# B&R Automation Studio project AnsteuerungSchrittmotor
Automation Studio 4.3.7.46 SP; technology packages: Acp10Arnc0 3.18.2

## Configuration Config1

CPU 4PP065.0571-P74, AutomationRuntime G4.34, Build 4.1.2, Vc V4.34.3

### Hardware
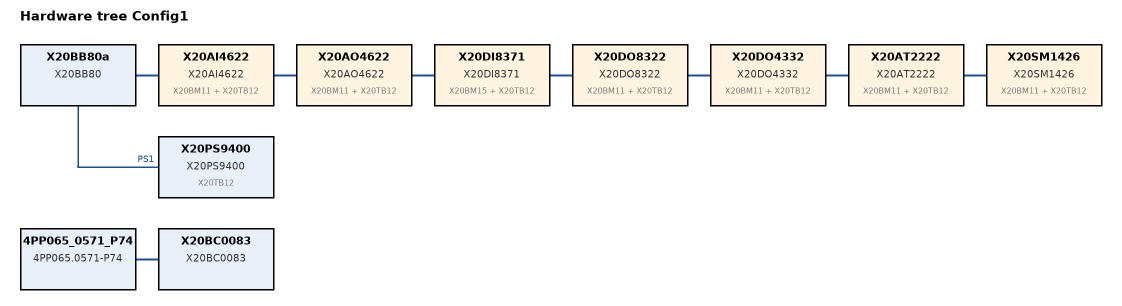
```
4PP065_0571_P74 : 4PP065.0571-P74 v1.1.2.0
  Connector IF5:
    ActivateDevice = 1
    Mode = Manual
    InternetAddress = 10.100.85.8
    SubnetMask = 255.255.255.0
  ConfigurationID = KainerKerschbaumer_Config1
  TimerDeviceType = EPLX2X
  TimerDevice = 4PP065_0571_P74.IF4
  TaskClassIdleTime = 2000
  Cyclic1Duration = 2000
  Cyclic1Tolerance = 0
  Cyclic1Output = 1
  VcObjectName = Visu
X20AI4622 : X20AI4622 v1.0.4.0  [SS1 -> X20TB12.SS; SL -> X20BM11.SL1]
X20AO4622 : X20AO4622 v1.1.0.0  [SS1 -> X20TB12e.SS; SL -> X20BM11c.SL1]
X20AT2222 : X20AT2222 v1.2.1.0  [SS1 -> X20TB12f.SS; SL -> X20BM11d.SL1]
X20BB80a : X20BB80 v1.0.1.0
X20BC0083 : X20BC0083 v2.5.3.0  [PLK1 -> 4PP065_0571_P74.IF4 (NodeNumber=1) [Cable Type=PowerlinkCable, Length=10, Version=1.0.0.1]; SL -> X20BB80a.SL1]
X20BM11 : X20BM11 v1.0.0.1  [X2X1 -> X20BB80a.IF1]
X20BM11a : X20BM11 v1.0.0.1  [X2X1 -> X20BM15.X2X2]
X20BM11b : X20BM11 v1.0.0.1  [X2X1 -> X20BM11a.X2X2]
X20BM11c : X20BM11 v1.0.0.1  [X2X1 -> X20BM11.X2X2]
X20BM11d : X20BM11 v1.0.0.1  [X2X1 -> X20BM11b.X2X2]
X20BM11e : X20BM11 v1.0.0.1  [X2X1 -> X20BM11d.X2X2]
X20BM15 : X20BM15 v1.0.1.0  [X2X1 -> X20BM11c.X2X2 (NodeNumber=4)]
X20DI8371 : X20DI8371 v1.0.2.0  [SS1 -> X20TB12a.SS; SL -> X20BM15.SL1]
X20DO4332 : X20DO4332 v1.0.3.0  [SS1 -> X20TB12d.SS; SL -> X20BM11b.SL1]
X20DO8322 : X20DO8322 v1.0.2.0  [SS1 -> X20TB12c.SS; SL -> X20BM11a.SL1]
X20PS9400 : X20PS9400 v1.0.2.4  [SS1 -> X20TB12b.SS; PS -> X20BB80a.PS1]
X20SM1426 : X20SM1426 v1.5.1.1  [SS1 -> X20TB12g.SS; SL -> X20BM11e.SL1]
  HoldingCurrent = 60
  RatedCurrent = 80
  MaximumCurrent = 100
  LatchSync = Stepper latch value synchron (AB/R latch value asynchron)
  SCALE_ENCOD_INCR_r1 = 51200
  BothEndSwitchesAreNormallyOpen_r1 = on
  QuickStopIsNormallyOpen_r1 = on
X20TB12 : X20TB12 v1.0.0.0
X20TB12a : X20TB12 v1.0.0.0
X20TB12b : X20TB12 v1.0.0.0
X20TB12c : X20TB12 v1.0.0.0
X20TB12d : X20TB12 v1.0.0.0
X20TB12e : X20TB12 v1.0.0.0
X20TB12f : X20TB12 v1.0.0.0
X20TB12g : X20TB12 v1.0.0.0
```

### IoMap.iom - 4PP065_0571_P74/IoMap.iom
```iecst
VAR_CONFIG
	       Cyclic#1.gAxis01_DrvIf.iLifeCnt AT %IB."X20SM1426".LifeCnt;
	       Cyclic#1.gAxis01_DrvIf.iDrvOK AT %IX."X20SM1426".DrvOk01;
	       Cyclic#1.gAxis01_DrvIf.oBoostCurrent AT %QX."X20SM1426".BoostCurrent01;
	       Cyclic#1.gAxis01_DrvIf.oStandStillCurrent AT %QX."X20SM1426".StandstillCurrent01;
	       Cyclic#1.gAxis01_DrvIf.oSetTime AT %QW."X20SM1426".SetTime01;
	       Cyclic#1.gAxis01_MotorStep0 AT %QW."X20SM1426".Motor1Step0;
	       Cyclic#1.gAxis01_DiDoIf.iLifeCntDriveEnable AT %IB."X20SM1426".LifeCnt;
	       Cyclic#1.gAxis01_DiDoIf.iLifeCntDriveReady AT %IB."X20SM1426".LifeCnt;
	       Cyclic#1.gAxis01_DiDoIf.iDriveReady AT %IX."X20SM1426".DrvOk01;
	       Cyclic#1.gAxis01_DiDoIf.oDriveEnable AT %QX."X20SM1426".DriveEnable01;
	       Cyclic#1.gAxis01_EncIf1.iLifeCnt AT %IB."X20SM1426".LifeCnt;
	       Cyclic#1.gAxis01_EncIf1.iEncOK AT %IX."X20SM1426".EncOk01;
	       Cyclic#1.gAxis01_EncIf1.iActPos AT %IW."X20SM1426".ActPos01;
	       Cyclic#1.gAxis01_EncIf1.iRefPulsePos AT %IW."X20SM1426".RefPulsePos01;
	       Cyclic#1.gAxis01_EncIf1.iRefPulseCnt AT %IB."X20SM1426".RefPulseCnt01;
	       Cyclic#1.gAxis01_EncIf1.iActTime AT %IW."X20SM1426".ActTime01;
END_VAR
```

### Acp10cfg.ncc - 4PP065_0571_P74/Motion/Acp10cfg.ncc
```
NcConfiguration (Version=3.18.2, NcSwId=Acp10)
  ACP10CF1_typ:
    cnt_nettrc_rec_drive = 1500
    bufsize_trace_upload = 1200
    tc_nc_man_task = Cyclic #1
    glob_pv_as_ncobject = Yes
    ncsys_dl_broadcast = Yes
    ncsys_dl_acp_reset = Yes
    safemc_log_err_to_ax = Yes
    network_init:
      ncsw_init_execute = Yes
      automatic_execute = No
      node_nr_warning = Yes
      net_err_before_ncact = Yes
    nettrc:
      enter_parsecrec = Yes
      enter_ncaction = Yes
      save_ring_startidx = Yes
    cam_prof_download:
      cam_dat_dl_parallel = No
      tc_cam_dl_parallel = Task class for NC Manager task
    sdc_if[0]:
      if_name = SDC_IF1
      mc_broadcast_size = 800
      mc_broadcast_extdat = No
```

### Acp10map.ncm - 4PP065_0571_P74/Motion/Acp10map.ncm
```
NcMapping (NcSwId=Acp10)
  NcObject gAxis01 (ModuleId=X20SM1426, ModuleAddress=SDC_IF1.ST1, Type=ncAXIS, Channel=1, AcoposSimulation=Off, InitParameter=gAxis01i, AcoposParameter=gAxis01a, Disabled=FALSE, ModuleDisabled=FALSE)
```

## Logical view

Binary libraries used (declarations not repeated): operator, runtime, astime, AsIecCon, Acp10man 3.18.2, Acp10par 3.18.2, NcGlobal 3.18.2, Acp10sdc 3.18.2, Acp10_MC 3.18.2, brsystem, sys_lib, AsBrStr

### Global.var - Global variables
```iecst
VAR
	gAxis01 : ACP10AXIS_typ;
	gAxis01_HW : SdcHwCfg_typ := (0);
	gAxis01_DrvIf : SdcDrvIf16_typ := (0);
	gAxis01_EncIf1 : SdcEncIf16_typ := (0);
	gAxis01_DiDoIf : SdcDiDoIf_typ := (0);
	gAxis01_MotorStep0 : INT := (0);
END_VAR
```


### Program Logical/ncsdcctrl (IEC)

#### ncsdcctrlCyclic.st
```iecst
PROGRAM _CYCLIC

(* ### BEGIN gAxis01 ### *)

(* life counter emulation of digital inputs *)
       gAxis01_DiDoIf.iLifeCntReference := gAxis01_DiDoIf.iLifeCntReference + 1;
       gAxis01_DiDoIf.iLifeCntNegHwEnd  := gAxis01_DiDoIf.iLifeCntNegHwEnd  + 1;
       gAxis01_DiDoIf.iLifeCntPosHwEnd  := gAxis01_DiDoIf.iLifeCntPosHwEnd  + 1;

(* default function model of ACOPOSmicro: convert absolute steps to delta steps - overflow save delta calculation *)
       gAxis01_MotorStep0 := gAxis01_DrvIf.oSetPos - gAxis01_oSetPosOld;
       gAxis01_oSetPosOld := gAxis01_DrvIf.oSetPos;

(* ### END gAxis01 ### *)

END_PROGRAM
```

#### ncsdcctrlInit.st
```iecst
PROGRAM _INIT

(* ### BEGIN gAxis01 ### *)

(* initialize general interfaces *)
       gAxis01.size := gAxis01.size;
       gAxis01_HW.DrvIf_Typ := ncSDC_DRVSM16;
       brsstrcpy( ADR(gAxis01_HW.DrvIf_Name[0]), ADR('gAxis01_DrvIf') );
       gAxis01_HW.DiDoIf_Typ := ncSDC_DIDO;
       brsstrcpy( ADR(gAxis01_HW.DiDoIf_Name[0]), ADR('gAxis01_DiDoIf') );
       gAxis01_HW.EncIf1_Typ := ncSDC_ENC16;
       brsstrcpy( ADR(gAxis01_HW.EncIf1_Name[0]), ADR('gAxis01_EncIf1') );
       gAxis01_EncIf1.iLifeCnt := gAxis01_EncIf1.iLifeCnt;

(* initialize old-value for delta step calculation *)
       gAxis01_oSetPosOld := gAxis01_DrvIf.oSetPos;

(* ### END gAxis01 ### *)

END_PROGRAM
```

#### ncsdcctrl.var
```iecst
VAR
	gAxis01_oSetPosOld : INT := 0;
END_VAR
```

### Data object Logical/acp10etxde (Ett)

- acp10etxde.ett (not shown)

### Package Logical/gAxis01obj - gAxis01obj

### Data object Logical/gAxis01obj/gAxis01a (Apt)

#### gAxis01a.apt
```
AcoposParameterTable:
  Root Parameters:
    64232 = 51200 (Name=SM_SCALE_STEP)
    64233 = 1000 (Name=SM_SCALE_LOAD_UNITS)
    64234 = 1 (Name=SM_SCALE_LOAD_MOTREV)
    109 = 51200 (Name=SCALE_ENCOD_INCR)
```

### Data object Logical/gAxis01obj/gAxis01i (Ax)

#### gAxis01i.ax
```
InitParameter (Version=3.18.2, NcSwId=Acp10)
  ACP10AXIS_typ:
    dig_in:
      level:
        reference = ncACTIV_HI
        pos_hw_end = ncACTIV_HI
        neg_hw_end = ncACTIV_HI
        trigger1 = ncACTIV_HI
        trigger2 = ncACTIV_HI
    encoder_if:
      parameter:
        count_dir = ncSTANDARD
        scaling:
          load:
            units = 1000
            rev_motor = 1
    limit:
      parameter:
        v_pos = 10000
        v_neg = 10000
        a1_pos = 50000
        a2_pos = 50000
        a1_neg = 50000
        a2_neg = 50000
        t_jolt = 0
        t_in_pos = 0
        pos_sw_end = 2000000000
        neg_sw_end = -2000000000
        ds_warning = 500
        ds_stop = 1000
        a_stop = 1.0e30
        dv_stop = 0
        dv_stop_mode = ncOFF
    controller:
      mode = ncPOSITION
      position:
        kv = 50
        tn = 0
        t_predict = 0.01
        t_total = 0.01
        p_max = 1.0e30
        i_max = 0
      speed:
        kv = 2.0
        tn = 0
        t_filter = 0.0
        isq_filter1:
          type = ncOFF
          a0 = 0.0
          a1 = 0.0
          b0 = 0.0
          b1 = 0.0
          b2 = 0.0
          c0_par_id = 0
          c1_par_id = 0
        isq_filter2:
          type = ncOFF
          a0 = 0.0
          a1 = 0.0
          b0 = 0.0
          b1 = 0.0
          b2 = 0.0
          c0_par_id = 0
          c1_par_id = 0
        isq_filter3:
          type = ncOFF
          a0 = 0.0
          a1 = 0.0
          b0 = 0.0
          b1 = 0.0
          b2 = 0.0
          c0_par_id = 0
          c1_par_id = 0
      uf:
        type = ncLINEAR
        auto_config = ncMOTOR_PAR
        u0 = 0
        un = 0
        fn = 50.0
        k_f_slip = 0
      ff:
        torque_load = 0.0
        torque_pos = 0.0
        torque_neg = 0.0
        kv_torque = 0.0
        inertia = 0.0
        t_filter_a = 0.0
    move:
      stop:
        parameter[0]:
          decel_ramp = ncA_LIMIT
          controller = ncON
        parameter[1]:
          decel_ramp = ncA_LIMIT
          controller = ncON
        parameter[2]:
          decel_ramp = ncA_LIMIT
          controller = ncON
        parameter[3]:
          decel_ramp = ncA_LIMIT
          controller = ncON
        quickstop:
          decel_ramp = ncA_LIMIT
        drive_error:
          decel_ramp = ncA_LIMIT
      homing:
        parameter:
          s = 0
          v_switch = 5000
          v_trigger = 500
          a = 50000
          mode = ncDIRECT
          edge_sw = ncPOSITIVE
          start_dir = ncPOSITIVE
          trigg_dir = ncPOSITIVE
          ref_pulse = ncOFF
          fix_dir = ncOFF
          tr_s_block = 0
          torque_lim = 0
          ds_block = 0
          ds_stop = 0
      basis:
        parameter:
          v_pos = 5000
          v_neg = 5000
          a1_pos = 50000
          a2_pos = 50000
          a1_neg = 50000
          a2_neg = 50000
    message:
      text:
        parameter:
          format = ncBREAK
          columns = 80
          data_modul = acp10etxde
```

### Program Logical/LibACP10MC_SingleAx_ST/Basic (IEC) - Basic logical control

#### basicCyclic.st - cyclic code
```iecst
(********************************************************************
 * COPYRIGHT -- Bernecker + Rainer
 ********************************************************************
 * PROGRAM: Basic
 * File: basicCyclic.st
 * Author: Bernecker + Rainer
 * Created: December 01, 2009
 ********************************************************************
 * Implementation of Program Basic
 ********************************************************************)
PROGRAM _CYCLIC

(***************************************************************
        Control Sequence
***************************************************************)
(* status information is read before the step sequencer to attain a shorter reaction time *)
(************************ MC_READSTATUS *************************)
MC_ReadStatus_0.Enable := NOT(MC_ReadStatus_0.Error);
MC_ReadStatus_0.Axis := Axis1Obj;
MC_ReadStatus_0();
BasicControl.AxisState.Disabled             := MC_ReadStatus_0.Disabled;
BasicControl.AxisState.StandStill           := MC_ReadStatus_0.StandStill;
BasicControl.AxisState.Stopping             := MC_ReadStatus_0.Stopping;
BasicControl.AxisState.Homing               := MC_ReadStatus_0.Homing;
BasicControl.AxisState.DiscreteMotion       := MC_ReadStatus_0.DiscreteMotion;
BasicControl.AxisState.ContinuousMotion     := MC_ReadStatus_0.ContinuousMotion;
BasicControl.AxisState.SynchronizedMotion   := MC_ReadStatus_0.SynchronizedMotion;
BasicControl.AxisState.ErrorStop            := MC_ReadStatus_0.Errorstop;

(********************MC_BR_READDRIVESTATUS***********************)
MC_BR_ReadDriveStatus_0.Enable := NOT(MC_BR_ReadDriveStatus_0.Error);
MC_BR_ReadDriveStatus_0.Axis := Axis1Obj;
MC_BR_ReadDriveStatus_0.AdrDriveStatus := ADR(BasicControl.Status.DriveStatus);
MC_BR_ReadDriveStatus_0();

(******************** MC_READACTUALPOSITION *********************)
MC_ReadActualPosition_0.Enable := (NOT(MC_ReadActualPosition_0.Error));
MC_ReadActualPosition_0.Axis := Axis1Obj;
MC_ReadActualPosition_0();
IF(MC_ReadActualPosition_0.Valid = TRUE)THEN
    BasicControl.Status.ActPosition := MC_ReadActualPosition_0.Position;
END_IF

(******************** MC_READACTUALVELOCITY *********************)
MC_ReadActualVelocity_0.Enable := (NOT(MC_ReadActualVelocity_0.Error));
MC_ReadActualVelocity_0.Axis := Axis1Obj;
MC_ReadActualVelocity_0();
IF(MC_ReadActualVelocity_0.Valid = TRUE)THEN
    BasicControl.Status.ActVelocity := MC_ReadActualVelocity_0.Velocity;
END_IF

(************************ MC_READAXISERROR **********************)
MC_ReadAxisError_0.Enable := NOT(MC_ReadAxisError_0.Error);
MC_ReadAxisError_0.Axis := Axis1Obj;
MC_ReadAxisError_0.DataAddress := ADR(BasicControl.Status.ErrorText);
MC_ReadAxisError_0.DataLength := SIZEOF(BasicControl.Status.ErrorText);
MC_ReadAxisError_0.DataObjectName := 'acp10etxen';
MC_ReadAxisError_0();

(**************** CHECK FOR GENERAL AXIS ERROR ******************)
    IF ((MC_ReadAxisError_0.AxisErrorID <> 0) AND (MC_ReadAxisError_0.Valid = TRUE)) THEN
        AxisStep := STATE_ERROR_AXIS;
(***************** CHECK IF POWER SHOULD BE OFF *******************)
    ELSIF ((BasicControl.Command.Power = FALSE) AND (MC_ReadAxisError_0.Valid = TRUE)) THEN
        IF ((MC_ReadStatus_0.Errorstop = TRUE) AND (MC_ReadStatus_0.Valid = TRUE)) THEN
            AxisStep := STATE_ERROR_RESET;
        ELSE
            AxisStep := STATE_WAIT;
        END_IF
    END_IF

(* central monitoring OF stop command attains a shorter reaction TIME in CASE OF emergency stop *)
(******************CHECK FOR STOP COMMAND************************)
    IF (BasicControl.Command.Stop = TRUE) THEN
        IF ((AxisStep >= STATE_HOME) AND (AxisStep <= STATE_ERROR)) THEN
            (* reset all FB execute inputs we use *)
            MC_Home_0.Execute := 0;
            MC_Stop_0.Execute := 0;
            MC_MoveAbsolute_0.Execute := 0;
            MC_MoveAdditive_0.Execute := 0;
            MC_MoveVelocity_0.Execute := 0;
            MC_ReadAxisError_0.Acknowledge := 0;
            MC_Reset_0.Execute := 0;
            MC_Halt_0.Execute := 0;

            (* reset user commands *)
            BasicControl.Command.Halt := 0;
            BasicControl.Command.Home := 0;
            BasicControl.Command.MoveJogPos := 0;
            BasicControl.Command.MoveJogNeg := 0;
            BasicControl.Command.MoveVelocity := 0;
            BasicControl.Command.MoveAbsolute := 0;
            BasicControl.Command.MoveAdditive := 0;
            AxisStep := STATE_STOP;
        END_IF
    END_IF

CASE AxisStep OF

(******************** WAIT *************************)
    STATE_WAIT:  (* STATE: Wait *)
        IF (BasicControl.Command.Power = TRUE) THEN
            AxisStep := STATE_POWER_ON;
        ELSE
            MC_Power_0.Enable := FALSE;
        END_IF

        (* reset all FB execute inputs we use *)
        MC_Home_0.Execute := FALSE;
        MC_Stop_0.Execute := FALSE;
        MC_MoveAbsolute_0.Execute := FALSE;
        MC_MoveAdditive_0.Execute := FALSE;
        MC_MoveVelocity_0.Execute := FALSE;
        MC_Halt_0.Execute := FALSE;
        MC_ReadAxisError_0.Acknowledge := FALSE;
        MC_Reset_0.Execute := FALSE;

        (* reset user commands *)
        BasicControl.Command.Stop := FALSE;
        BasicControl.Command.Halt := FALSE;
        BasicControl.Command.Home := FALSE;
        BasicControl.Command.MoveJogPos := FALSE;
        BasicControl.Command.MoveJogNeg := FALSE;
        BasicControl.Command.MoveVelocity := FALSE;
        BasicControl.Command.MoveAbsolute := FALSE;
        BasicControl.Command.MoveAdditive := FALSE;

        BasicControl.Status.ErrorID := 0;

(******************** POWER ON **********************)
    STATE_POWER_ON:  (* STATE: Power on *)
        MC_Power_0.Enable := TRUE;
        IF (MC_Power_0.Status = TRUE) THEN
            AxisStep := STATE_READY;
        END_IF
        (* if a power error occured go to error state *)
        IF (MC_Power_0.Error = TRUE) THEN
            BasicControl.Status.ErrorID := MC_Power_0.ErrorID;
            AxisStep := STATE_ERROR;
        END_IF

(******************** READY **********************)
    STATE_READY:  (* STATE: Waiting for commands *)
        IF (BasicControl.Command.Home = TRUE)THEN
            BasicControl.Command.Home := FALSE;
            AxisStep := STATE_HOME;

        ELSIF (BasicControl.Command.Stop = TRUE) THEN
            AxisStep := STATE_STOP;

        ELSIF (BasicControl.Command.MoveJogPos = TRUE) THEN
            AxisStep := STATE_JOG_POSITIVE;

        ELSIF (BasicControl.Command.MoveJogNeg = TRUE) THEN
            AxisStep := STATE_JOG_NEGATIVE;

        ELSIF (BasicControl.Command.MoveAbsolute = TRUE) THEN
            BasicControl.Command.MoveAbsolute := FALSE;
            AxisStep := STATE_MOVE_ABSOLUTE;

        ELSIF (BasicControl.Command.MoveAdditive = TRUE) THEN
            BasicControl.Command.MoveAdditive := FALSE;
            AxisStep := STATE_MOVE_ADDITIVE;

        ELSIF (BasicControl.Command.MoveVelocity = TRUE) THEN
            BasicControl.Command.MoveVelocity := FALSE;
            AxisStep := STATE_MOVE_VELOCITY;

        ELSIF (BasicControl.Command.Halt = TRUE) THEN
            BasicControl.Command.Halt := FALSE;
            AxisStep := STATE_HALT;
        END_IF

(******************** HOME **********************)
    STATE_HOME:  (* STATE: start homing process *)
        MC_Home_0.Position := BasicControl.Parameter.HomePosition;
        MC_Home_0.HomingMode := BasicControl.Parameter.HomeMode;
        MC_Home_0.Execute := TRUE;
        IF (MC_Home_0.Done = TRUE) THEN
            MC_Home_0.Execute := FALSE;
            AxisStep := STATE_READY;
        END_IF
        (* if a homing error occured go to error state *)
        IF (MC_Home_0.Error = TRUE) THEN
            MC_Home_0.Execute := FALSE;
            BasicControl.Status.ErrorID := MC_Home_0.ErrorID;
            AxisStep := STATE_ERROR;
        END_IF

(***********************HALT_MOVEMENT***************************)
    STATE_HALT:   (* STATE: Halt movement *)
        MC_Halt_0.Deceleration := BasicControl.Parameter.Deceleration;
        MC_Halt_0.Execute := TRUE;
        IF (MC_Halt_0.Done = TRUE) THEN
            MC_Halt_0.Execute := FALSE;
            AxisStep := STATE_READY;
        END_IF
        (* check if error occured *)
        IF (MC_Halt_0.Error = TRUE) THEN
            BasicControl.Status.ErrorID := MC_Halt_0.ErrorID;
            MC_Halt_0.Execute := FALSE;
            AxisStep := STATE_ERROR;
        END_IF

(*********************** STOP MOVEMENT *************************)
    STATE_STOP:  (* STATE: Stop movement *)
        MC_Stop_0.Deceleration := BasicControl.Parameter.Deceleration;
        MC_Stop_0.Execute := TRUE;
        (* if axis is stopped go to ready state *)
        IF ((MC_Stop_0.Done = TRUE) AND (BasicControl.Command.Stop = FALSE)) THEN
            MC_Stop_0.Execute := FALSE;
            AxisStep := STATE_READY;
        END_IF
        (* check if error occured *)
        IF (MC_Stop_0.Error = TRUE) THEN
            BasicControl.Status.ErrorID := MC_Stop_0.ErrorID;
            MC_Stop_0.Execute := FALSE;
            AxisStep := STATE_ERROR;
        END_IF

(******************** START JOG MOVEMENT POSITVE **********************)
     STATE_JOG_POSITIVE:  (* STATE: Start jog movement in positive direction *)
        MC_MoveVelocity_0.Velocity      := BasicControl.Parameter.JogVelocity;
        MC_MoveVelocity_0.Acceleration  := BasicControl.Parameter.Acceleration;
        MC_MoveVelocity_0.Deceleration  := BasicControl.Parameter.Deceleration;
        MC_MoveVelocity_0.Direction     := mcPOSITIVE_DIR;
        MC_MoveVelocity_0.Execute := TRUE;
        IF (BasicControl.Command.MoveJogPos = FALSE) THEN
            MC_MoveVelocity_0.Execute := FALSE;
            AxisStep := STATE_HALT;
        END_IF
        (* check if error occured *)
        IF (MC_MoveVelocity_0.Error = TRUE) THEN
            BasicControl.Status.ErrorID := MC_MoveVelocity_0.ErrorID;
            MC_MoveVelocity_0.Execute := FALSE;
            AxisStep := STATE_ERROR;
        END_IF

(******************** START JOG MOVEMENT NEGATIVE **********************)
    STATE_JOG_NEGATIVE:  (* STATE: Start jog movement in negative direction *)
        MC_MoveVelocity_0.Velocity      := BasicControl.Parameter.JogVelocity;
        MC_MoveVelocity_0.Acceleration  := BasicControl.Parameter.Acceleration;
        MC_MoveVelocity_0.Deceleration  := BasicControl.Parameter.Deceleration;
        MC_MoveVelocity_0.Direction	    := mcNEGATIVE_DIR;
        MC_MoveVelocity_0.Execute := TRUE;
        IF (BasicControl.Command.MoveJogNeg = FALSE) THEN
            MC_MoveVelocity_0.Execute := FALSE;
            AxisStep := STATE_HALT;
        END_IF
        (* check if error occured *)
        IF (MC_MoveVelocity_0.Error = TRUE) THEN
            BasicControl.Status.ErrorID := MC_MoveVelocity_0.ErrorID;
            MC_MoveVelocity_0.Execute := FALSE;
            AxisStep := STATE_ERROR;
        END_IF

(******************** START ABSOLUTE MOVEMENT **********************)
     STATE_MOVE_ABSOLUTE:  (* STATE: Start absolute movement *)
        MC_MoveAbsolute_0.Position      := BasicControl.Parameter.Position;
        MC_MoveAbsolute_0.Velocity      := BasicControl.Parameter.Velocity;
        MC_MoveAbsolute_0.Acceleration  := BasicControl.Parameter.Acceleration;
        MC_MoveAbsolute_0.Deceleration  := BasicControl.Parameter.Deceleration;
        MC_MoveAbsolute_0.Direction     := BasicControl.Parameter.Direction;
        MC_MoveAbsolute_0.Execute := TRUE;
        (* check if commanded position is reached *)
        IF (BasicControl.Command.Halt) THEN
            BasicControl.Command.Halt := FALSE;
            MC_MoveAbsolute_0.Execute := FALSE;
            AxisStep := STATE_HALT;
        ELSIF (MC_MoveAbsolute_0.Done = TRUE) THEN
            MC_MoveAbsolute_0.Execute := FALSE;
            AxisStep := STATE_READY;
        END_IF
        (* check if error occured *)
        IF (MC_MoveAbsolute_0.Error = TRUE) THEN
            BasicControl.Status.ErrorID := MC_MoveAbsolute_0.ErrorID;
            MC_MoveAbsolute_0.Execute := FALSE;
            AxisStep := STATE_ERROR;
        END_IF

(******************** START ADDITIVE MOVEMENT **********************)
    STATE_MOVE_ADDITIVE:  (* STATE: Start additive movement *)
        MC_MoveAdditive_0.Distance      := BasicControl.Parameter.Distance;
        MC_MoveAdditive_0.Velocity      := BasicControl.Parameter.Velocity;
        MC_MoveAdditive_0.Acceleration  := BasicControl.Parameter.Acceleration;
        MC_MoveAdditive_0.Deceleration  := BasicControl.Parameter.Deceleration;
        MC_MoveAdditive_0.Execute := TRUE;
        (* check if commanded distance is reached *)
        IF (BasicControl.Command.Halt) THEN
            BasicControl.Command.Halt := FALSE;
            MC_MoveAdditive_0.Execute := FALSE;
            AxisStep := STATE_HALT;
        ELSIF (MC_MoveAdditive_0.Done = TRUE) THEN
            MC_MoveAdditive_0.Execute := FALSE;
            AxisStep := STATE_READY;
        END_IF
        (* check if error occured *)
        IF (MC_MoveAdditive_0.Error = TRUE) THEN
            BasicControl.Status.ErrorID := MC_MoveAdditive_0.ErrorID;
            MC_MoveAdditive_0.Execute := FALSE;
            AxisStep := STATE_ERROR;
        END_IF

(******************** START VELOCITY MOVEMENT **********************)
    STATE_MOVE_VELOCITY:  (* STATE: Start velocity movement *)
        MC_MoveVelocity_0.Velocity      := BasicControl.Parameter.Velocity;
        MC_MoveVelocity_0.Acceleration  := BasicControl.Parameter.Acceleration;
        MC_MoveVelocity_0.Deceleration  := BasicControl.Parameter.Deceleration;
        MC_MoveVelocity_0.Direction     := BasicControl.Parameter.Direction;
        MC_MoveVelocity_0.Execute := TRUE;
        (* check if commanded velocity is reached *)
        IF (BasicControl.Command.Halt) THEN
            BasicControl.Command.Halt := FALSE;
            MC_MoveVelocity_0.Execute := FALSE;
            AxisStep := STATE_HALT;
        ELSIF (MC_MoveVelocity_0.InVelocity = TRUE) THEN
            MC_MoveVelocity_0.Execute := FALSE;
            AxisStep := STATE_READY;
        END_IF
        (* check if error occured *)
        IF (MC_MoveVelocity_0.Error = TRUE) THEN
            BasicControl.Status.ErrorID := MC_MoveVelocity_0.ErrorID;
            MC_MoveVelocity_0.Execute := FALSE;
            AxisStep := STATE_ERROR;
        END_IF

(******************** FB-ERROR OCCURED *************************)
    STATE_ERROR:  (* STATE: Error *)
        (* check if FB indicates an axis error *)
        IF (MC_ReadAxisError_0.AxisErrorCount<>0) THEN
            AxisStep := STATE_ERROR_AXIS;
        ELSE
            IF (BasicControl.Command.ErrorAcknowledge = TRUE) THEN
                BasicControl.Command.ErrorAcknowledge := FALSE;
                BasicControl.Status.ErrorID := 0;
                (* reset axis if it is in axis state ErrorStop *)
                IF ((MC_ReadStatus_0.Errorstop = TRUE) AND (MC_ReadStatus_0.Valid = TRUE)) THEN
                    AxisStep := STATE_ERROR_RESET;
                ELSE
                    AxisStep := STATE_WAIT;
                END_IF
            END_IF
        END_IF

(******************** AXIS-ERROR OCCURED *************************)
    STATE_ERROR_AXIS:  (* STATE: Axis Error *)
        IF (MC_ReadAxisError_0.Valid = TRUE) THEN
            IF (MC_ReadAxisError_0.AxisErrorID <> 0) THEN
                BasicControl.Status.ErrorID := MC_ReadAxisError_0.AxisErrorID;
            END_IF
            MC_ReadAxisError_0.Acknowledge := FALSE;
            IF (BasicControl.Command.ErrorAcknowledge = TRUE) THEN
                BasicControl.Command.ErrorAcknowledge := FALSE;
                (* acknowledge axis error *)
                IF (MC_ReadAxisError_0.AxisErrorID <> 0) THEN
                    MC_ReadAxisError_0.Acknowledge := TRUE;
                END_IF
            END_IF
            IF (MC_ReadAxisError_0.AxisErrorCount = 0) THEN
                (* reset axis if it is in axis state ErrorStop *)
                BasicControl.Status.ErrorID := 0;
                IF ((MC_ReadStatus_0.Errorstop = TRUE) AND (MC_ReadStatus_0.Valid = TRUE)) THEN
                    AxisStep := STATE_ERROR_RESET;
                ELSE
                    AxisStep := STATE_WAIT;
                END_IF
            END_IF
        END_IF

(******************** RESET DONE *************************)
    STATE_ERROR_RESET:  (* STATE: Wait for reset done *)
        MC_Reset_0.Execute := TRUE;
        (* reset MC_Power.Enable if this FB is in Error*)
        IF (MC_Power_0.Error = TRUE) THEN
            MC_Power_0.Enable := FALSE;
        END_IF
        IF(MC_Reset_0.Done = TRUE)THEN
            MC_Reset_0.Execute := FALSE;
            AxisStep := STATE_WAIT;
        ELSIF(MC_Reset_0.Error = TRUE) THEN
            MC_Reset_0.Execute := FALSE;
            AxisStep := STATE_ERROR;
        END_IF
(******************** SEQUENCE END *************************)
END_CASE

(***************************************************************
        Function Block Calls
***************************************************************)

(************************** MC_POWER ****************************)
MC_Power_0.Axis := Axis1Obj;  (* pointer to axis *)
MC_Power_0();

(************************** MC_HOME *****************************)
MC_Home_0.Axis := Axis1Obj;
MC_Home_0();

(********************** MC_MOVEABSOLUTE *************************)
MC_MoveAbsolute_0.Axis := Axis1Obj;
MC_MoveAbsolute_0();

(********************** MC_MOVEADDITIVE *************************)
MC_MoveAdditive_0.Axis := Axis1Obj;
MC_MoveAdditive_0();

(********************** MC_MOVEVELOCITY *************************)
MC_MoveVelocity_0.Axis := Axis1Obj;
MC_MoveVelocity_0();

(************************** MC_STOP *****************************)
MC_Stop_0.Axis := Axis1Obj;
MC_Stop_0();

(***************************MC_HALT******************************)
MC_Halt_0.Axis := Axis1Obj;
MC_Halt_0();

(************************** MC_RESET ****************************)
MC_Reset_0.Axis := Axis1Obj;
MC_Reset_0();

END_PROGRAM
```

#### basicInit.st - init code
```iecst
PROGRAM _INIT

(* get axis object *)
Axis1Obj := ADR(gAxis01);

AxisStep := STATE_WAIT; (* start step *)

BasicControl.Parameter.Velocity             := 1000;  (*velocity for movement*)
BasicControl.Parameter.Acceleration         := 5000;  (*acceleration for movement*)
BasicControl.Parameter.Deceleration         := 5000;  (*deceleration for movement*)
BasicControl.Parameter.JogVelocity          := 400;   (*velocity for jogging *)
END_PROGRAM
```

#### basic.typ - Local data types
```iecst
TYPE
	basic_command_typ : 	STRUCT  (*command structure*)
		Power : BOOL; (*switch on the controller*)
		Home : BOOL; (*reference the axis*)
		MoveAbsolute : BOOL; (*move to an defined position*)
		MoveAdditive : BOOL; (*move a defiened distance*)
		MoveVelocity : BOOL; (*start a movement with a defiened velocity*)
		Halt : BOOL; (*stop every active movement*)
		Stop : BOOL; (*stop every active movement as long as is set*)
		MoveJogPos : BOOL; (*move in positive direction as long as is set*)
		MoveJogNeg : BOOL; (*move in negative direction as long as is set*)
		ErrorAcknowledge : BOOL; (*reset active errors*)
	END_STRUCT;
	basic_parameter_typ : 	STRUCT  (*parameter structure*)
		Position : REAL; (*target-position for MoveAbsolute-Command*)
		Distance : REAL; (*distance for MoveAdditive-Command*)
		Velocity : REAL; (*velocity for MoveVelocity-Command*)
		Direction : USINT; (*direction for commanded movements*)
		Acceleration : REAL; (*acceleration for commanded movements*)
		Deceleration : REAL; (*deceleration for commanded movements*)
		HomePosition : REAL; (*target-position for referencing the axis*)
		HomeMode : USINT; (*homing mode*)
		JogVelocity : REAL; (*velocity for jogging movement*)
	END_STRUCT;
	basic_status_typ : 	STRUCT  (*status structure*)
		ErrorID : UINT; (*ErrorID of any occured error*)
		ErrorText : ARRAY[0..3] OF STRING[79]; (*Error Text*)
		ActPosition : REAL; (*actual position of the axis*)
		ActVelocity : REAL; (*actual velocity of the axis*)
		DriveStatus : MC_DRIVESTATUS_TYP; (*actual status of the axis*)
	END_STRUCT;
	basic_axisState_typ : 	STRUCT  (*axis state structure*)
		Disabled : BOOL; (*if set, axis is in state Disabled*)
		StandStill : BOOL; (*if set, axis is in state StandsStill*)
		Homing : BOOL; (*if set, axis is in state Homing*)
		Stopping : BOOL; (*if set, axis is in state Stopping*)
		DiscreteMotion : BOOL; (*if set, axis is in state DiscreteMotion*)
		ContinuousMotion : BOOL; (*if set, axis is in state ContinousMotion*)
		SynchronizedMotion : BOOL; (*if set, axis is in state SynchronizedMotion*)
		ErrorStop : BOOL; (*if set, axis is in state ErrorStop*)
	END_STRUCT;
	basic_typ : 	STRUCT  (*control structure*)
		Command : basic_command_typ; (*command structure*)
		Parameter : basic_parameter_typ; (*parameter structure*)
		Status : basic_status_typ; (*status structure*)
		AxisState : basic_axisState_typ; (*axis state structure*)
	END_STRUCT;
END_TYPE
```

#### basic.var - Local variables
```iecst
VAR
	BasicControl : basic_typ; (*control structure*)
	MC_Home_0 : MC_Home; (*Function Block*)
	MC_MoveAbsolute_0 : MC_MoveAbsolute; (*Function Block*)
	MC_MoveAdditive_0 : MC_MoveAdditive; (*Function Block*)
	MC_MoveVelocity_0 : MC_MoveVelocity; (*Function Block*)
	MC_Power_0 : MC_Power; (*Function Block*)
	MC_ReadActualPosition_0 : MC_ReadActualPosition; (*Function Block *)
	MC_ReadActualVelocity_0 : MC_ReadActualVelocity; (*Function Block*)
	MC_ReadAxisError_0 : MC_ReadAxisError; (*Function Block*)
	MC_ReadStatus_0 : MC_ReadStatus; (*Function Block*)
	MC_Reset_0 : MC_Reset; (*Function Block*)
	MC_Stop_0 : MC_Stop; (*Function Block*)
	MC_BR_ReadDriveStatus_0 : MC_BR_ReadDriveStatus; (*Function Block*)
	MC_Halt_0 : MC_Halt; (*Function Block*)
	Axis1Obj : UDINT; (*axis reference*)
	AxisStep : UINT; (*current step in the step sequence*)
END_VAR
VAR CONSTANT
	STATE_READY : USINT := 10; (*constant for a waiting step*)
	STATE_POWER_ON : USINT := 1; (*constant for the step in which the controller is switched on*)
	STATE_MOVE_VELOCITY : USINT := 16; (*constant for the step in which a movement with defiened velocity is started*)
	STATE_MOVE_ABSOLUTE : USINT := 14; (*constant for the step in which a movement to defiened position is started*)
	STATE_WAIT : USINT := 0; (*constant for a waiting step*)
	STATE_STOP : USINT := 11; (*constant for the step in which movements are stopped*)
	STATE_MOVE_ADDITIVE : USINT := 15; (*constant for the step in which a movement with defiened distance is started*)
	STATE_HOME : USINT := 2; (*constant for the step in which the axis is homed*)
	STATE_ERROR_RESET : USINT := 102; (*constant for the step in which the errors are reset*)
	STATE_ERROR_AXIS : USINT := 100; (*constant for the axis error step*)
	STATE_ERROR : USINT := 101; (*constant for the error step*)
	STATE_JOG_POSITIVE : USINT := 12; (*constant for the step in which a positive jogging movement is executed*)
	STATE_JOG_NEGATIVE : USINT := 13; (*constant for the step in which a negative jogging movement is executed*)
	STATE_HALT : USINT := 17; (*constant for the step in which movements are stopped*)
END_VAR
```

- Visualisation Logical/Visu (not shown)

Listed in the project but not available here: Logical/Global.typ, Logical/ncsdcctrl/ncsdcctrl.typ
